(*

.. <legal notes>

legal notes
=================
| SPDX-FileCopyrightText: © 2026 Oleksandr Tiutyk <trofimich@gmail.com>
| SPDX-License-Identifier: LGPL-3.0-only
| For details check: LGPL-3.0-only_

.. _LGPL-3.0-only: https://www.gnu.org/licenses/lgpl-3.0.en.html

.. </legal notes>

*)

FUNCTION_BLOCK RangeInt32AnalogValueConverter EXTENDS Core.Object IMPLEMENTS IAnalogValueConverter
VAR_OUTPUT
	MinDigitizedValue : DINT;
	MaxDigitizedValue : DINT;
	MinPhysicalValue : LREAL;
	MaxPhysicalValue : LREAL;
END_VAR
VAR
	_ClassName : STRING := __POUNAME();
END_VAR

{attribute 'monitoring' := 'call'}
PROPERTY ClassName : STRING
GET
ClassName := _ClassName;
END_GET
END_PROPERTY

METHOD ConvertAnalogValueToDigitizedValue : DIGITIZED_ANALOG_VALUE
VAR_INPUT
	analogValue	: LREAL;
END_VAR
IF analogValue >= MaxPhysicalValue THEN
	ConvertAnalogValueToDigitizedValue._32Bit := MaxDigitizedValue;
ELSIF analogValue <= MinPhysicalValue THEN
	ConvertAnalogValueToDigitizedValue._32Bit := MinDigitizedValue;
ELSE
    ConvertAnalogValueToDigitizedValue._32Bit := TO_DINT((analogValue - MinPhysicalValue) / (MaxPhysicalValue - MinPhysicalValue) * TO_LREAL(MaxDigitizedValue - MinDigitizedValue) + TO_LREAL(MinDigitizedValue));
END_IF
END_METHOD

METHOD ConvertDigitizedValueToAnalogValue : LREAL
VAR_INPUT
	digitizedValue : DIGITIZED_ANALOG_VALUE;
END_VAR
IF digitizedValue._32Bit= MaxDigitizedValue THEN
	ConvertDigitizedValueToAnalogValue := MaxPhysicalValue;
ELSIF digitizedValue._32Bit = MinDigitizedValue THEN
	ConvertDigitizedValueToAnalogValue := MinPhysicalValue;
ELSE
	ConvertDigitizedValueToAnalogValue := TO_LREAL(digitizedValue._32Bit - MinDigitizedValue) / TO_LREAL(MaxDigitizedValue - MinDigitizedValue) * (MaxPhysicalValue - MinPhysicalValue) + MinPhysicalValue;
END_IF
END_METHOD

METHOD FB_init : BOOL
VAR_INPUT
	(* if TRUE, the retain variables are initialized (warm start / cold start)*)
	bInitRetains	: BOOL;
	(* if TRUE, the instance afterwards gets moved into the copy code (online change)*)
	bInCopyCode	: BOOL;
	minDigitizedValue : DINT;
	maxDigitizedValue : DINT;
	minPhysicalValue : LREAL;
	maxPhysicalValue : LREAL;
END_VAR
THIS^.MinDigitizedValue := minDigitizedValue;
THIS^.MaxDigitizedValue := maxDigitizedValue;
THIS^.MinPhysicalValue := minPhysicalValue;
THIS^.MaxPhysicalValue := maxPhysicalValue;
END_METHOD

{attribute 'monitoring' := 'call'}
PROPERTY NamespaceName : STRING
GET
NamespaceName := CurrentNamespace.Name;
END_GET
END_PROPERTY

{attribute 'monitoring' := 'call'}
PROPERTY SelfSize : ULINT
GET
SelfSize := XSIZEOF(THIS^);
END_GET
END_PROPERTY

END_FUNCTION_BLOCK

(* stored: Version 1.1.0.1
   POU RangeInt32AnalogValueConverter: Id {8635bf3a-7ddb-4863-847d-060b4774f236}, SpecialFunc None
   Property ClassName: Id {2605209c-aa5d-48f1-b5a5-feff1831541d}
   Get Get: Id {9ebe162b-ff33-4714-8269-d56b870ef8ba}
   Method ConvertAnalogValueToDigitizedValue: Id {ce161fc1-4794-449b-a925-96878b653591}
   Method ConvertDigitizedValueToAnalogValue: Id {c70aaedc-168c-428c-913b-72f86c123b1b}
   Method FB_init: Id {6e528392-d48d-4cff-9a21-af8cc61754e4}
   Property NamespaceName: Id {a54ed07f-fbe1-41b5-b5e5-6d50d9fb54b9}
   Get Get: Id {ef8c248a-3c4a-4fbe-be30-475fcbb83200}
   Property SelfSize: Id {188fe25d-c91b-4d47-a0c2-a9833a8525bc}
   Get Get: Id {eeaf7768-e212-4a49-8505-97c7a06613c1} *)
